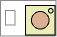
VISUALIZATION VISU_SafetyEmergencyStop  // 57x37
VAR_IN_OUT
	contactNC : BOOL;
    contactNO : BOOL;
END_VAR
    Rectangle (25,5 30x30)
    Frame (5,10 10x15)
        shows VISU_State_red_green(state := contactNC)
    Ellipse (31,11 18x18)
    Ellipse (48,8 5x5), colour toggle: contactNO
END_VISUALIZATION

(* stored: Version 1.1.0.1, ProductVersion 3.1.4019.2
   Visu VISU_SafetyEmergencyStop: Id {9ee7b87c-ea37-4d49-89da-5819c8f60f5c} *)
